PROGRAM MAIN
VAR
	fHysteresis: REAL := 1;
	fbSR: SR;
END_VAR
VAR // added by the converter: edge detectors and wires of the graphical bodies
    _w1, _w2 : ANY;
END_VAR

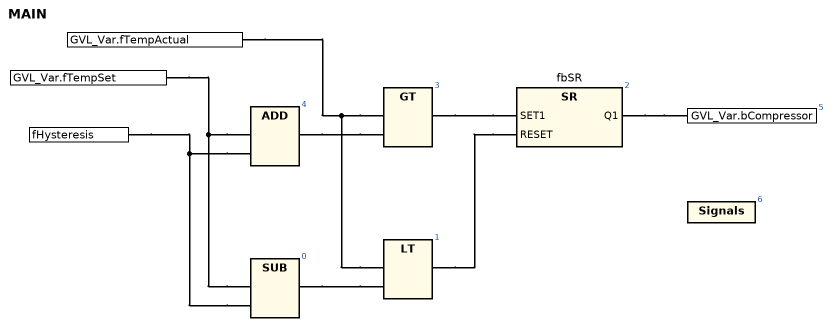
fbSR(SET1 := _w1, RESET := GVL_Var.fTempActual < GVL_Var.fTempSet - fHysteresis); // SR
_w1 := GVL_Var.fTempActual > _w2;
_w2 := GVL_Var.fTempSet + fHysteresis;
GVL_Var.bCompressor := fbSR.Q1;
Signals();

END_PROGRAM

(* stored: Version 1.1.0.1, ProductVersion 3.1.4024.4
   POU MAIN: Id {239fa1f1-b9a5-4096-9e50-7c1f215c2670}, SpecialFunc None *)
